(* CoDeSys 2.3.9.62 project: Semaforo11_7.pro *)
(* Libraries: Standard.lib 2.6.14 10:37:46, IecSfc.lib 2.6.14 11:37:46 *)

(* Global variable list: Global_Variables *)
VAR_GLOBAL

 (* Entradas *)
	M: BOOL;

      (*Salidas*)
	Rojo: BOOL;    	(* Luz roja*)
	Amarillo:BOOL;	(* Luz amarilla *)
	Verde:BOOL;		(* Luz verde *)

      (* CONTADOR *)
      Conta:CTU;

END_VAR

(* POU PLC_PRG, LD *)
PROGRAM PLC_PRG
VAR

END_VAR
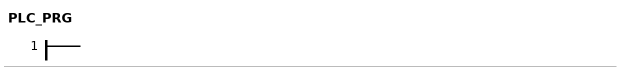
_LD_ (* Ladder Diagram *)
NETWORK 1
	*
_END_LD_
(* the same logic as Structured Text *)
(* Network 1 *)
END_PROGRAM

(* POU AccionConta, LD *)
PROGRAM AccionConta
VAR
END_VAR
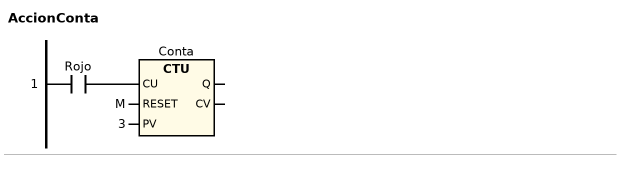
_LD_ (* Ladder Diagram *)
NETWORK 1
	[Rojo] - Conta:CTU(CU: *, RESET: M, PV: 3)
_END_LD_
(* the same logic as Structured Text *)
(* Network 1 *)
Conta(CU := Rojo, RESET := M, PV := 3);
END_PROGRAM

(* POU ControlSemaforo, SFC *)
PROGRAM ControlSemaforo
VAR
END_VAR
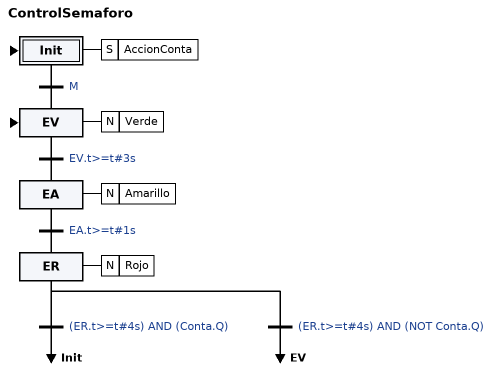
INITIAL_STEP Init:
	AccionConta(S);
END_STEP
TRANSITION FROM Init TO EV := M;
END_TRANSITION
STEP EV:
	Verde(N);
END_STEP
TRANSITION FROM EV TO EA := EV.t>=t#3s;
END_TRANSITION
STEP EA:
	Amarillo(N);
END_STEP
TRANSITION FROM EA TO ER := EA.t>=t#1s;
END_TRANSITION
STEP ER:
	Rojo(N);
END_STEP
TRANSITION FROM ER TO Init := (ER.t>=t#4s) AND (Conta.Q);
END_TRANSITION
TRANSITION FROM ER TO EV := (ER.t>=t#4s) AND (NOT Conta.Q);
END_TRANSITION
END_PROGRAM

(* Visualisation SemaforoSimple
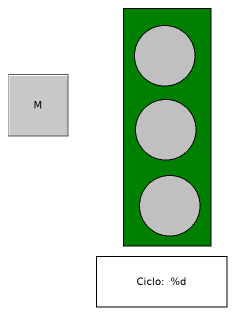
ellipse at (156,41)-(217,102): alarm colour if Rojo
ellipse at (157,115)-(218,176): alarm colour if Amarillo
ellipse at (161,191)-(222,252): alarm colour if Verde
rectangle at (118,272)-(249,323): text "Ciclo:  %d"; shows CONTA.CV
button at (30,90)-(90,152): text "M"; taps M
1 more shapes without text or variables
*)
